FUNCTION_BLOCK S5Gate
  (* Standard: 61499-2 *)
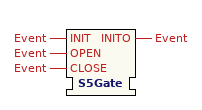
  EVENT_INPUT
    INIT;
    OPEN;
    CLOSE;
  END_EVENT
  EVENT_OUTPUT
    INITO;
  END_EVENT
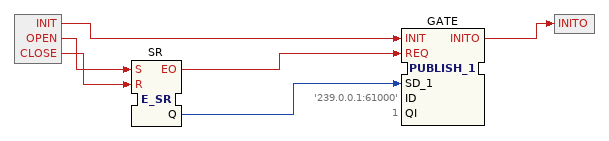
  FBS
    SR : E_SR;
    GATE : PUBLISH_1(ID := '239.0.0.1:61000', QI := 1);
  END_FBS
  EVENT_CONNECTIONS
    OPEN TO SR.S;
    CLOSE TO SR.R;
    INIT TO GATE.INIT;
    SR.EO TO GATE.REQ;
    GATE.INITO TO INITO;
  END_CONNECTIONS
  DATA_CONNECTIONS
    SR.Q TO GATE.SD_1;
  END_CONNECTIONS
END_FUNCTION_BLOCK
